(* CODESYS project CAN API.library
   Author: 3S - Smart Software Solutions GmbH
   Title: CAN API
   Version: 1.0.0.3
   DocFormat: reStructuredText
   Description: This library provides an easy to use interface for sending and receiving CAN messages. The library is optimized for Structured Text and graphical (CFC) programming.
   Company: 3S - Smart Software Solutions GmbH
   LanguageModelAttribute: qualified-access-only
   DefaultNamespace: CAN

Project tree, tasks and I/O mapping:
  libraries: CAA Behaviour Model, * (CAA Technical Workgroup); CANbus, * (3S - Smart Software Solutions GmbH); CAA Memory Block Manager Extern, * (CAA Technical Workgroup); Standard, * (System)
  Enums/
    data type RECEIVERTYPE
    data type BUSSTATE
    data type ERROR
  Interfaces/
    interface IMessageProcessor: ProcessMessage
    interface ICANBus29bit
    interface ICANDriver: ICANBus
    interface ICANBusBase: GetBusDiagnosis, DeleteReceiver, GetAreaReceiver, ReceiveMessage, SendMessage, ResetBusAlarm, CloseCANDriver, Is29bit, GetMaskReceiver, GetSingleIdReceiver
    interface ICANBus11bit
  00000000-0000-0000-0000-000000000000|D:\CoDeSys\LibrariesV3\trunk\Intern\CAA\CAA Template\3.4.0.0 draft\Placeholder.xml
  00000000-0000-0000-0000-000000000000|D:\CoDeSys\LibrariesV3\trunk\Intern\CAA\CAA Template\3.2.0.3 draft\Prefix.pdf
  Function Blocks/
    Object Oriented Programming/
      function block CANBus_11bit [ST]: GetBusDiagnosis, Is29bit, ResetBusAlarm, ReceiveMessage, CloseCANDriver, DeleteReceiver, GetMaskReceiver, GetAreaReceiver, GetSingleIdReceiver, SendMessage
      function block CANBus_Base [ST]: CloseCANDriver, SendMessage, DeleteReceiver, FreeReceiverBlock, ReceiveAlwaysNewest, GetReceiverBlock, CreateMaskReceiver, CreateAreaReceiver, ReceiveQueued, CreateSingleIDReceiver, CreateDriver, BusAlarm, GetAreaReceiver, GetMaskReceiver, ReceiveMessage, FB_Init, GetBusDiagnosis, ResetBusAlarm, Is29bit, GetSingleIdReceiver
      function block CANBus_29bit [ST]: ResetBusAlarm, SendMessage, DeleteReceiver, GetMaskReceiver, ReceiveMessage, Is29bit, CloseCANDriver, GetAreaReceiver, GetBusDiagnosis, GetSingleIdReceiver
    Graphical Programming/
      function block CANSender [ST]: prvAbort, prvResetOutputs, prvStart, prvCyclicAction
      function block CANBusDiagnosis [ST]: prvResetOutputs, prvCyclicAction, prvStart, prvAbort
      function block CANDriver_11bit [ST]: ICANBus, prvCyclicAction, prvAbort, prvStart, prvResetOutputs
      function block CANAreaReceiver [ST]: prvAbort, prvCyclicAction, prvResetOutputs, prvStart
      function block CANDriver_29bit [ST]: ICANBus, prvCyclicAction, prvResetOutputs, prvStart, prvAbort
      function block CANMaskReceiver [ST]: prvStart, prvAbort, prvCyclicAction, prvResetOutputs
      function block CANSingleIdReceiver [ST]: prvResetOutputs, prvStart, prvAbort, prvCyclicAction
  Structs/
    data type RECEIVER_INFO
    data type DRIVER_CONFIG
    data type RECEIVER_MASK
    data type MESSAGE
    data type RxMESSAGE
    data type RECEIVER_AREA
    data type DIAGNOSIS_INFO
    data type RECEIVER_SINGLE_ID
*)

// Structs/RECEIVER_INFO
{attribute 'hide'}
{attribute 'qualified_only'}
TYPE RECEIVER_INFO :
STRUCT
	hReceiver : CAA.HANDLE;
	eType : RECEIVERTYPE;
END_STRUCT
END_TYPE

// Structs/DRIVER_CONFIG
/// This data type describes the configuration of a CANbus Driver
{attribute 'qualified_only'}
TYPE DRIVER_CONFIG :
STRUCT
	uiBaudrate 		: UINT; (* Possible values for baud rate [kbit/s]: 10, 20, 50, 100, 125, 250, 500, 800 or 1000. *)
	usiNetwork 		: USINT; (* number of the interface (Network ID starts by 0) *)
	ctMessages		: USINT; (* length of the message queue for outgoing messages *)
END_STRUCT
END_TYPE

// Structs/RECEIVER_MASK
/// | The parameter canIdMask describes a bit mask for canId’s on incoming messages. 
/// | The parameter canIdValue proofs if the mask applies to the CanId of the received message. 
/// | If the CanId doesn’t apply to the mask, the message will be filtered out. 
/// | For the use of the other Mask/Value parameters see the examples of RECEIVER_AREA.
{attribute 'qualified_only'}

TYPE RECEIVER_MASK :
STRUCT
	dwIdValue 			: DWORD; (* bit sign of identifier of message *)
	dwIdMask 			: DWORD; (* mask for bit sign of IdValue *)
	xRTRValue 			: BOOL; (* bit sign for RTR flag *)
	xRTRMask 			: BOOL; (* mask for bit sign of xRTRValue  *)
	x29BitIdValue 		: BOOL; (* 29-Bit message *)
	x29BitIdMask 		: BOOL; (* Mask for 29-bit message *)
	xTransmitValue 		: BOOL; (* Messages sent via this adapter with the same driver. *)
	xTransmitMask 		: BOOL; (* Mask for messages sent via this adapter with the same driver. *)
	xAlwaysNewest 		: BOOL; (* TRUE: only the most current message will be received; FALSE: all messages will be received *)
END_STRUCT
END_TYPE

// Enums/RECEIVERTYPE
/// | This data type distinguishes if a receiver receives always the newest message or not  
{attribute 'qualified_only'}
TYPE RECEIVERTYPE :
(
	QUEUED_RECEIVER, (* receiving all messages *)
	ALWAYS_NEWEST_RECEIVER (* receiving only the newest message *)
) BYTE;
END_TYPE

// Enums/BUSSTATE
/// | This data type describes the current state of the CAN network.
{attribute 'qualified_only'}
TYPE BUSSTATE :
(
	UNKNOWN := 0, (* The state of the network is not known. Its functionality is not implemented. *)
	ERR_FREE, (* No occurrence of CAN bus errors so far. The error counters of the chip are zero. *)
	ACTIVE, (* Only few CAN bus errors so far. The error counters of the chip are below the warning level. *)
	WARNING, (* Occurrence of some CAN bus errors. The error counters are above the warning level. *)
	PASSIVE, (* Too many CAN bus errors. The error counters are above the error level. *)
	BUSOFF (* The node has been separated from the CAN bus. The error counter has exceeded the admissible maximum. *)
)BYTE;
END_TYPE

// Structs/MESSAGE
/// | This structure contains the information of a message. 
/// | Messages of this type can be sent via CANSender (FB) in CFC or by an instance of CANBus_11bit / CANBus_29bit  
/// | in ST programs.
{attribute 'qualified_only'}
TYPE MESSAGE :
STRUCT
	udiCanID 		: UDINT; (* CAN-ID (Communication Object Identifier) is the bitId of a CAN-frame *)
	abyData 		: ARRAY[0..7] OF BYTE; (* Array for 0 to 7 bytes of data *)
	usiDataLength 	: USINT; (* The length of the data array 0 to 8 *)
	xRTR 			: BOOL; (* Remote Transmission Request *)
	xIs29BitMessage	: BOOL; (* TRUE: the messages is a 29bit message, FALSE: the message is a 11bit message *)
END_STRUCT
END_TYPE

// Structs/RxMESSAGE
/// | The structure of a received message. RxMESSAGE has two more elements as MESSAGE.
/// | Messages of the type RxMESSAGE can be used the same way as messages of the type MESSAGE
{attribute 'qualified_only'}
TYPE RxMESSAGE EXTENDS MESSAGE :
STRUCT
		xIsTxMessage	: BOOL := TRUE; (* TRUE: Messages sent via this adapter with the same driver. *)
		udiTSP			: UDINT; (* Only available if the driver supports TimeStamps. If not the value is 0. Compare TimeStamp by calling SysTimeGetUs() function *)
END_STRUCT
END_TYPE

// Structs/RECEIVER_AREA
/// | This structure identifies an area for receiving CANBus frames. 
/// | Please note that the Area Receiver only allows 11bit CAN-IDs. If the mask parameter is TRUE, 
/// | a filter in the CAN Receiver Queue is active. 
/// | Now messages are filtered according to the value parameter. 
/// |
/// | Examples:
/// | Only Transmit messages ranging between 16#100 and 16#150: 
/// | dwIdStart:=16#100, dwIdEnd:=16#150, xTransmitValue = TRUE, xTransmitMask = TRUE, all other Mask paramters = FALSE
/// |
/// | All messages ranging between 16#0 and 16#7FF 
/// | dwIdStart:=16#0, dwIdEnd:=16#7FF all mask parameters FALSE (no further filtering is done).
/// |
/// | All messages: dwIdStart = 0, dwIdEnd = 0, 
/// | all Mask Parameter FALSE all Value Parameter FALSE
/// |
{attribute 'qualified_only'}
TYPE RECEIVER_AREA :
STRUCT
	dwIdStart		: DWORD; (* first identifier of the area *)
	dwIdEnd			: DWORD; (* last identifier of the area *)
	xRTRValue		: BOOL; (* bit sign for RTR flag *)
	xRTRMask		: BOOL; (* mask for bit sign of xRTRValue  *)
	xTransmitValue	: BOOL; (* Messages sent via this adapter with the same driver. *)
	xTransmitMask	: BOOL; (* Mask for messages sent via this adapter with the same driver. *)
END_STRUCT
END_TYPE

// Structs/DIAGNOSIS_INFO
/// This data type describes diagnostic information 
{attribute 'qualified_only'}
TYPE DIAGNOSIS_INFO :
STRUCT
	ctSendCounter			: CAA.COUNT; (* The value of the send counter. *)
	ctReceiveCounter		: CAA.COUNT; (* The value of the receive counter. *)
	ctRxErrorCounter		: CAA.COUNT; (* The value of the receive error counter. *)
	ctTxErrorCounter		: CAA.COUNT; (* The value of the send error counter. *)	
	ctLostCounter			: CAA.COUNT; (* The value of the lost messages. *)
	ctReceivePoolSize		: CAA.COUNT; (* Size of the receive pool *)
	ctReceiveQueueLength	: CAA.COUNT; (* Size of the receive queue length *)
	ctTransmitPoolSize		: CAA.COUNT; (* Size of the transmit pool *)
	ctTransmitQueueLength	: CAA.COUNT; (* Size of the transmit queue length *)
	xBusAlarm				: BOOL; (* Bus Alarm *)
	usiBusLoad				: USINT; (* The bus load. *)
	xSendingActive			: BOOL; (*  TRUE: the CAN hardware is busy sending CAN messages. FALSE: all messages have already been sent. *)
	eState					: BUSSTATE; (* This data type describes the state of the CAN network. *)
	uiBaudrate				: UINT; (* The baud rate of the bus. *)
END_STRUCT
END_TYPE

// Enums/ERROR
/// | This data type describes errors
{attribute 'qualified_only'}
TYPE ERROR : 
(
		NO_ERROR := 0, (* No error occurred *)
		INTERNAL_ERROR, (* An error occurred in the CL2 Library. Please check with brake points. *)
		NO_MEMORY, (* no more memory *)
		NO_CANBUS_DRIVER, (* Create a valid CANBus Driver for this operation *)
		NO_VALID_RECEIVER, (* There is no valid receiver *)
		START_VALUE_GT_END, (* Start value is greater than end value for area receiver *)
		TIME_OUT, (* Time out *)
		BUS_ALARM, (* The CAN Bus is in alarm state *)
		MESSAGE_QUEUE_EXCEEDED, (* The sending queue is full *)
		ONLY_11BIT_CANID_ALLOWED, (* CAN-IDs needs to be max. 11bit *)
		WRONG_BAUDRATE, (* Baudrate for CANDriver is not valid *)
		WRONG_PARAMETER, (* A parameter has a wrong value *)
		CANBUS_DRIVER_NOT_CREATED (* NetID might be wrong or the driver is not registered in "GatewayPLC/CoDeSysControl.cfg".
									Example 1: 1 CAN card with 2 channels, channel 1: NetId = 0, channel 2: NetId = 1;
									Example 2: 2 CAN cards: NetId depends on the order the drivers are loaded. *) 
)BYTE; 
END_TYPE

// Structs/RECEIVER_SINGLE_ID
/// | This structure filters the messages of a single CAN Id. 
/// | If the mask parameter is TRUE, a filter in the CAN Receiver Queue is active. 
/// | Now messages are filtered according to the value parameter. Also see the examples of RECEIVER_AREA.
{attribute 'qualified_only'}
TYPE RECEIVER_SINGLE_ID :
STRUCT
	dwCanId			: DWORD; (* CanId *)
	xRTRValue		: BOOL; (* bit sign for RTR flag *)
	xRTRMask		: BOOL; (* mask for bit sign of xRTRValue  *)
	x29BitIdValue	: BOOL; (* 29-Bit message *)
	x29BitIdMask	: BOOL; (* Mask for 29-bit message *)
	xTransmitValue	: BOOL; (* Messages sent via this adapter with the same driver. *)
	xTransmitMask	: BOOL; (* Mask for messages sent via this adapter with the same driver. *)
	xAlwaysNewest	: BOOL; (* TRUE: only the most current message will be received; FALSE: all messages will be received *)
END_STRUCT
END_TYPE

// Interfaces/IMessageProcessor
/// All received messages are passed to the MessageProcessor. The method ProcessMessage() must be implemented by the user.
INTERFACE IMessageProcessor

/// | The Process Message Method must be implemented by the user.
/// | Define here how you wish to proceed with incoming messages.
METHOD ProcessMessage
VAR_IN_OUT
	Message 		: RxMESSAGE; (* Incoming message *)
END_VAR
END_METHOD

END_INTERFACE

// Interfaces/ICANBus29bit
{attribute 'hide'}
INTERFACE ICANBus29bit EXTENDS ICANBusBase

END_INTERFACE

// Interfaces/ICANBusBase
{attribute 'hide'}
INTERFACE ICANBusBase EXTENDS __SYSTEM.IQueryInterface

METHOD GetBusDiagnosis : BOOL
VAR_IN_OUT
	DiagnosticInfo		: DIAGNOSIS_INFO; (* This data type descripes diagnostic information  *)
END_VAR
VAR_OUTPUT
	eError				: ERROR; (* Error codes *)
END_VAR
END_METHOD

METHOD DeleteReceiver : BOOL
VAR_IN_OUT
	hReceiver		: CAA.HANDLE; (* Receiver to be deleted *)
END_VAR
VAR_OUTPUT
	eError			: ERROR; (* Error codes *)
END_VAR
END_METHOD

METHOD GetAreaReceiver : CAA.HANDLE
VAR_IN_OUT
	Area				: RECEIVER_AREA; (* Structure with the information of the bit masks and a range of CAN-IDs *)
END_VAR
VAR_OUTPUT
	eError				: ERROR; (* Error codes *)
END_VAR
END_METHOD

METHOD ReceiveMessage : BOOL
VAR_INPUT
	hReceiver 		: CAA.HANDLE; (* Eather a MaskReceiver or AreaReceiver *)
	itfMsgProcessor : IMessageProcessor;
	tTimeLimit		: TIME;
END_VAR
VAR_OUTPUT
	eError			: ERROR; (* Error codes *)
END_VAR
END_METHOD

METHOD SendMessage : BOOL
VAR_IN_OUT
	Message 		: Message; (* Structure with the frame information and data to be sent. *)
END_VAR
VAR_OUTPUT
	eError			: ERROR; (* Error codes *)
END_VAR
END_METHOD

METHOD ResetBusAlarm : BOOL
VAR_INPUT
END_VAR
VAR_OUTPUT
	eError			: ERROR; (* Error codes *)
END_VAR
END_METHOD

METHOD CloseCANDriver : BOOL
VAR_OUTPUT
	eError			: ERROR; (* Error codes *)
END_VAR
END_METHOD


PROPERTY Is29bit : BOOL
GET
END_GET
END_PROPERTY

METHOD GetMaskReceiver : CAA.HANDLE
VAR_IN_OUT
	Mask				: RECEIVER_MASK; (* Structure with the information of the bit masks *)
END_VAR
VAR_OUTPUT
	eError				: ERROR; (* Error codes *)
END_VAR
END_METHOD

METHOD GetSingleIdReceiver : CAA.HANDLE
VAR_IN_OUT
	SingleId			: RECEIVER_SINGLE_ID; (* Structure with the information of the bit masks *)
END_VAR
VAR_OUTPUT
	eError				: ERROR; (* Error codes *)
END_VAR
END_METHOD

END_INTERFACE

// Function Blocks/Graphical Programming/CANSender
/// | CANSender will send messages over a CANDriver. It is possible to send frames with 29 bit and 11 bit frames. 
/// | This depends on the CAN Driver used for instantiating the CAN Sender. A CAN Sender instantiated with a 29BitCANDriver 
/// | is able to send 11 bit messages as well as 29 bit messages. The sending method is defined by 
/// | setting the xSendAs29bitMsg flag of MESSAGE. An 11BitCANDriver can only send 11 bit messages. 
/// | If CANSender uses an 11bit driver xSendAs29bitMsg of MESSAGE will be ignored.
FUNCTION_BLOCK CANSender EXTENDS CBM.ETrig
VAR_INPUT
	itfCANDriver	: ICANDriver; (* Messages are sent with this driver *)
END_VAR
VAR_IN_OUT
	Message 		: MESSAGE; (* Message information and data. *)
END_VAR
VAR_OUTPUT
	eError			: ERROR; (* Error codes *)
END_VAR
VAR
	_itf11bit			: ICANBus11bit;
	_itf29bit			: ICANBus29bit;
	_hReceiver			: CAA.HANDLE;
	_pMessage 			: POINTER TO MESSAGE;
END_VAR

_pMessage := ADR(Message);
SUPER^();

{attribute 'hide'}
METHOD prvAbort : BOOL
VAR_INPUT
END_VAR
VAR
END_VAR
(*IF xError THEN (* abort because of error *)

ELSE (* user abort *)

END_IF*)
xAbortInProgress:= FALSE;
END_METHOD

{attribute 'hide'}
METHOD prvResetOutputs : BOOL
VAR_INPUT
END_VAR
VAR
END_VAR
eError:= ERROR.NO_ERROR;
SUPER^.prvResetOutputs();
END_METHOD

{attribute 'hide'}
METHOD prvStart : BOOL
VAR_INPUT
END_VAR
VAR
END_VAR
END_METHOD

{attribute 'hide'}
METHOD prvCyclicAction : BOOL
VAR_INPUT
END_VAR
VAR
END_VAR
IF _pMessage <> CAA.gc_pNULL THEN
	IF (itfCANDriver.ICANBus.Is29bit) THEN
		__QUERYINTERFACE(itfCANDriver.ICANBus, _itf29Bit);
		_itf29bit.SendMessage(Message:=_pMessage^, eError=>eError);
	ELSE
		__QUERYINTERFACE(itfCANDriver.ICANBus, _itf11Bit);
		_itf11bit.SendMessage(Message:=_pMessage^, eError=>eError);
	END_IF
END_IF

IF eError = ERROR.NO_ERROR THEN
	xDone:= TRUE;
ELSE
	iError:= 2;
END_IF
END_METHOD

END_FUNCTION_BLOCK

// Interfaces/ICANDriver
/// | CANDriver_11bit and CANDriver_29bit implement this interface. 
/// | CANSender, CANMaskReceiver, CANAreaReceiver and CANBusDiagnosis expect a CANDriver instance that implements 
/// | the ICANDriver interface.
INTERFACE ICANDriver

{attribute 'hide'}
PROPERTY ICANBus : ICANBusBase
GET
END_GET
END_PROPERTY

END_INTERFACE

// Function Blocks/Graphical Programming/CANDriver_11bit
/// | This CAN Driver can handle frames with 11bit CAN-IDs. If a CAN Sender gets instantiated with this Driver all messages
/// | are sent in 11 bit frames. The xSendAs29bitMsg flag of Message will be ignored. Any Receiver instantiated with this Driver
/// | will only receive frames with 11 bit CAN-IDs. In case of a Bus Alarm it’s possible to reset the driver through xResetBusAlarm.
FUNCTION_BLOCK CANDriver_11bit EXTENDS CBM.LTrig IMPLEMENTS ICANDriver
VAR_INPUT
	xResetBusAlarm	: BOOL; (* TRUE: Reset the Bus Alarm (applies only if the Bus Driver is in alarm state). *)
END_VAR
VAR_IN_OUT
	DriverConfig	: DRIVER_CONFIG; (* Information to setup the CANbus Driver *)
END_VAR
VAR_OUTPUT
	xBusAlarm		: BOOL; (* Indicates if a Bus Alarm occurred *)
	eError			: ERROR; (* Error codes *)
END_VAR
VAR
	_CANBus			: CANBus_11bit;
	_pDriverConfig	: POINTER TO DRIVER_CONFIG;
END_VAR

_pDriverConfig := ADR(DriverConfig);
SUPER^();
IF iError = CBM.ERROR.TIME_OUT THEN
	eError := ERROR.TIME_OUT;
END_IF

{attribute 'hide'}
PROPERTY ICANBus : ICANBusBase
GET
ICANBus:= _CANBus;
END_GET
END_PROPERTY

{attribute 'hide'}
METHOD prvCyclicAction : BOOL
VAR_INPUT
END_VAR
VAR
END_VAR
IF xEnable AND _pDriverConfig <> CAA.gc_pNULL THEN
	_CANBus(DriverConfig:= _pDriverConfig^, eError=> eError);
	IF _CANBus.BusAlarm THEN 
		eError:= ERROR.BUS_ALARM;
		xBusAlarm:= TRUE;
	ELSIF (*_CANBus.BusAlarm AND*) xResetBusAlarm  THEN
		_CANBus.ResetBusAlarm(eError=> eError);
		xBusAlarm:= FALSE;
	END_IF
END_IF

IF eError <> ERROR.NO_ERROR THEN
	iError:= 2;
END_IF
END_METHOD

{attribute 'hide'}
METHOD prvAbort : BOOL
VAR_INPUT
END_VAR
VAR
END_VAR
IF xError THEN (* abort because of error *)
	_CANBus.CloseCANDriver(eError=> eError);
ELSE
	_CANBus.CloseCANDriver(eError=> eError);
END_IF
xAbortInProgress:= FALSE;
END_METHOD

{attribute 'hide'}
METHOD prvStart : BOOL
VAR_INPUT
END_VAR
VAR
END_VAR
END_METHOD

{attribute 'hide'}
METHOD prvResetOutputs : BOOL
VAR_INPUT
END_VAR
VAR
END_VAR
eError:= ERROR.NO_ERROR;
xBusAlarm:= FALSE;
SUPER^.prvResetOutputs();
END_METHOD

END_FUNCTION_BLOCK

// Function Blocks/Object Oriented Programming/CANBus_11bit
/// | CANBus_11bit can handle frames with 11bit CAN-IDs. An instance of this function block has to be created in order 
/// | for being able to send or receive messages. The FB expects a complete structure of the type DRIVER_CONFIG 
/// | to set up the CANBus.
FUNCTION_BLOCK CANBus_11bit EXTENDS CANBus_Base IMPLEMENTS ICANBus11bit
VAR_INPUT
END_VAR
VAR_OUTPUT
END_VAR
VAR
END_VAR

/// Call of the CANBus_Base FB
SUPER^._x29bitSupport:= FALSE;
SUPER^();

/// This method aggregates diagnostic information in DIAGNOSIS_INFO 
METHOD GetBusDiagnosis : BOOL
VAR_IN_OUT
	DiagnosticInfo		: DIAGNOSIS_INFO; (* This data type descripes diagnostic information  *)
END_VAR
VAR_OUTPUT
	eError				: ERROR; (* Error codes *)
END_VAR
/// Method call of the CANBus_Base FB
GetBusDiagnosis:= SUPER^.GetBusDiagnosis(DiagnosticInfo:= DiagnosticInfo, eError=> eError);
END_METHOD

{attribute 'hide'}
PROPERTY Is29bit : BOOL
GET
Is29bit:= FALSE;
END_GET
END_PROPERTY

/// This method resets the CANBus if the driver is in 'bus alarm' state. 
METHOD ResetBusAlarm : BOOL
VAR_INPUT
END_VAR
VAR_OUTPUT
	eError			: ERROR; (* Error codes *)
END_VAR
/// Method call of the CANBus_Base FB
ResetBusAlarm:= SUPER^.ResetBusAlarm(eError=> eError);
END_METHOD

/// | ReceiveMessage expects a valid handle to either an AreaReceiver, SingleIdReceiver or a MaskReceiver. 
/// | With receivers it is possible to filter incoming messages. If a time limit is set, the receiver will 
/// | receive in each cycle messages until the time is up. It there is no time limit set (tTimeLimit:= 0), 
/// | the receiver receives messages until the receiver buffer is empty. If the time limit is too small it 
/// | may be that not all received messages are processed and therefor the buffer gets smaller until there 
/// | are no free message handles left. Received messages will be passed to the Message Processor. All message 
/// | information will be available there. The Message Processor must be implemented by the user.
METHOD ReceiveMessage : BOOL
VAR_INPUT
	hReceiver 		: CAA.HANDLE; (* Either a MaskReceiver, SingleIdReceiver or AreaReceiver *)
	itfMsgProcessor : IMessageProcessor; (* The Message Processor will process the read messages accrding to the implementation of the user *)
	tTimeLimit		: TIME; (* The time limit for reading messages. (T#0s means no time limit) *)
END_VAR
VAR_OUTPUT
	eError			: ERROR; (* Error codes *)
END_VAR
/// Method call of the CANBus_Base FB
ReceiveMessage:= SUPER^.ReceiveMessage(hReceiver:= hReceiver, itfMsgProcessor:= itfMsgProcessor, tTimeLimit:= tTimeLimit, eError=> eError);
END_METHOD

/// | Closes the CAN Driver. After closing, messages can't be received or transmitted anymore.
METHOD CloseCANDriver : BOOL
VAR_INPUT
END_VAR
VAR_OUTPUT
	eError			: ERROR; (* Error codes *)
END_VAR
CloseCANDriver:= SUPER^.CloseCANDriver(eError=> eError);
END_METHOD

/// Deletes given receiver
METHOD DeleteReceiver : BOOL
VAR_IN_OUT
	hReceiver		: CAA.HANDLE; (* Receiver to be deleted *)
END_VAR
VAR_IN_OUT
END_VAR
VAR_OUTPUT
	eError			: ERROR; (* Error codes *)
END_VAR
/// Method call of the CANBus_Base FB
DeleteReceiver:= super^.DeleteReceiver(hReceiver:= hReceiver, eError=> eError);
END_METHOD

/// | Creates a mask for receiving messages. (With each call of this function a Receiver is created. 
/// | Therefor the method should not be called cyclic.)
METHOD GetMaskReceiver : CAA.HANDLE
VAR_IN_OUT
	Mask				: RECEIVER_MASK; (* Structure with the information of the bit masks *)
END_VAR
VAR_OUTPUT
	eError				: ERROR; (* Error codes *)
END_VAR
/// Method call of the CANBus_Base FB
GetMaskReceiver:= SUPER^.GetMaskReceiver(Mask:= Mask, eError=> eError);
END_METHOD

/// | Creates a receiver to receive messages within a range of CAN-IDs. 
/// | (With each call of this function a Receiver is created. Therefor the method should not be called cyclic.)
METHOD GetAreaReceiver : CAA.HANDLE
VAR_IN_OUT
	Area				: RECEIVER_AREA; (* Structure with the information of the bit masks and a range of CAN-IDs *)
END_VAR
VAR_OUTPUT
	eError				: ERROR; (* Error codes *)
END_VAR
/// Method call of the CANBus_Base FB
GetAreaReceiver:= SUPER^.GetAreaReceiver(Area:= Area, eError=> eError);
END_METHOD

/// | Generates a receiver for filtering a single CanId. (With each call of this function a 
/// | Receiver is created. Therefor the method should not be called cyclic.)
METHOD GetSingleIdReceiver : CAA.HANDLE
VAR_IN_OUT
	(* Structure with the information of the bit masks *)
	SingleId	: RECEIVER_SINGLE_ID;
END_VAR
VAR_OUTPUT
	(* Error codes *)
	eError	: ERROR;
END_VAR
/// Method call of the CANBus_Base FB
GetSingleIdReceiver:= SUPER^.GetSingleIdReceiver(SingleId:= SingleId, eError=> eError);
END_METHOD

/// Send a message. If the message got sent the return value is true.
METHOD SendMessage : BOOL
VAR_IN_OUT
	Message 		: MESSAGE; (* Message information and data. *)
END_VAR
VAR_OUTPUT
	eError			: ERROR; (* Error codes *)
END_VAR
SendMessage := SUPER^.SendMessage(Message := Message, eError => eError);
END_METHOD

END_FUNCTION_BLOCK

// Function Blocks/Object Oriented Programming/CANBus_Base
/// This is the base function block for CANBus_11bit and CANBus_29bit
{attribute 'hide'}
FUNCTION_BLOCK CANBus_Base IMPLEMENTS ICANBusBase
VAR_INPUT
	DriverConfig	: DRIVER_CONFIG; (* This structure contains the informaiton for creating a CANbus Driver *)
END_VAR
VAR_OUTPUT
	eError			: ERROR; (* Error codes *)
END_VAR
VAR
	_hDriver			: CAA.HANDLE; (* The handle for the CANbus Driver *)
	_hReceiverPool		: CAA.HANDLE;
	_x29bitSupport	: BOOL;
	_eErrorInternal	: CL2.ERROR; (* error codes from the CL2 library *)
END_VAR

/// By calling the private method CreateDriver() a CANbus Driver will be created. The driver is accessable through hDriver.
IF _hDriver = CAA.gc_hINVALID THEN
	CreateDriver(DriverConfig:= DriverConfig, x29bitSupport:= _x29bitSupport, hDriver=> _hDriver, eError=> eError);
END_IF

/// Closes the CAN Driver. After closing, messages can't be received or transmitted anymore.
METHOD CloseCANDriver : BOOL
VAR_INPUT
END_VAR
VAR_OUTPUT
	eError			: ERROR; (* Error codes *)
END_VAR
VAR
	eErrorInternal	: CL2.ERROR; (* error codes from the CL2 library *)
END_VAR
IF _hDriver <> CAA.gc_hINVALID THEN
	eErrorInternal:= CL2.DriverClose(hDriver:= _hDriver);
	IF eErrorInternal <> CL2.ERROR.NO_ERROR THEN
		eError:= ERROR.INTERNAL_ERROR;
	ELSE
		_hDriver:= CAA.gc_hINVALID;
		CloseCANDriver:= TRUE;
	END_IF
ELSE
	eError:= ERROR.NO_CANBUS_DRIVER;
END_IF
END_METHOD

/// Send a message. If the message got sent the return value is true.
METHOD SendMessage : BOOL
VAR_IN_OUT
	Message 		: MESSAGE; (* Message information and data. *)
END_VAR
VAR_OUTPUT
	eError			: ERROR; (* Error codes *)
END_VAR
VAR
	hMessage		: CAA.HANDLE; (* Pointer to the created Message *)
	eErrorInternal	: CL2.ERROR; (* error codes from the CL2 library *)
	pData			: POINTER TO CL2i.DATA; (* Pointer to the data array of the created message *)
	i				: INT; (* Counter *)
END_VAR
IF(_hDriver <> CAA.gc_hINVALID)THEN
	IF NOT Is29Bit AND MESSAGE.xIs29BitMessage THEN
		eError := ERROR.ONLY_11BIT_CANID_ALLOWED;
		RETURN;
	END_IF
	
	IF NOT Message.xIs29BitMessage THEN
		IF Message.udiCanID > 16#7FF THEN
			eError := ERROR.WRONG_PARAMETER;
			RETURN;
		END_IF
	END_IF
	
	/// First it creates a new message with the data from Message by calling CL2.CreateMessage()
	hMessage:= CL2.CreateMessage(
				hDriver:= _hDriver, 
				cobID:= Message.udiCanId, 
				usiLength:= Message.usiDataLength, 
				xRTR:= Message.xRTR, 
				x29BitID:= Message.xIs29BitMessage,
				peError:= ADR(eErrorInternal));

	IF hMessage <> CAA.gc_hINVALID THEN
		IF Message.usiDataLength > 0 THEN
			/// The data from the data-array will be copied into the data-array of the created message			
			pData:= CL2.GetMessageDataPointer(hMessage:= hMessage, peError:= ADR(eErrorInternal));
			FOR i:=0 TO Message.usiDataLength -1 DO
				pData^[i]:= Message.abyData[i];
			END_FOR
		END_IF
		
		/// The frame with the data is sent when CL2.Write() gets called.			
		eErrorInternal := CL2.Write(hDriver:= _hDriver, hMessage:= hMessage, usiPriority:= 2, xEnableSyncWindow:= FALSE);
		IF eErrorInternal <> CL2.ERROR.NO_ERROR THEN
			eError:= ERROR.INTERNAL_ERROR;
			IF hMessage <> CAA.gc_hINVALID THEN
				CL2.FreeMessage(hMessage:= hMessage);
				hMessage := CAA.gc_hINVALID;
			END_IF
		ELSE
			SendMessage:= TRUE;
		END_IF
	ELSE
		eError:= ERROR.MESSAGE_QUEUE_EXCEEDED;
	END_IF
ELSE
	eError:= ERROR.NO_CANBUS_DRIVER;
END_IF
END_METHOD

/// Deletes any receiver
METHOD DeleteReceiver : BOOL
VAR_IN_OUT
	hReceiver		: CAA.HANDLE; (* Receiver to be deleted *)
END_VAR
VAR_IN_OUT
END_VAR
VAR_OUTPUT
	eError			: ERROR; (* Error codes *)
END_VAR
VAR
	pReceiverInfo : POINTER TO RECEIVER_INFO;
	eErrorInternal	: CL2.ERROR; (* error codes from the CL2 library *)
	eMBMError : MBM.ERROR;
END_VAR
IF hReceiver <> CAA.gc_hINVALID THEN
	pReceiverInfo := MBM.BlockGetData(hBlock := hReceiver, peError := ADR(eMBMError));
	IF pReceiverInfo <> CAA.gc_pNULL THEN
		eErrorInternal:= CL2.DeleteReceiver(hReceiverId:= pReceiverInfo^.hReceiver);
		pReceiverInfo^.hReceiver := CAA.gc_hINVALID;
		MBM.PoolPutBlock(hReceiver);
		DeleteReceiver:= TRUE;
	ELSE
		eError:= ERROR.NO_VALID_RECEIVER;
	END_IF
ELSE
	eError:= ERROR.NO_VALID_RECEIVER;
END_IF
END_METHOD

METHOD PRIVATE FreeReceiverBlock
VAR_INPUT
	hReceiverBlock : CAA.HANDLE;
END_VAR
VAR
END_VAR
MBM.PoolPutBlock(hBlock := hReceiverBlock);
END_METHOD

METHOD PRIVATE ReceiveAlwaysNewest : BOOL
VAR_INPUT	
	hReceiver 		: CAA.HANDLE; (* Eather a MaskReceiver or AreaReceiver *)
	itfMsgProcessor : IMessageProcessor; (* The Message Processor will process the read messages accrding to the implementation of the user *)
END_VAR
VAR_OUTPUT
	eError			: ERROR; (* Error codes *)
END_VAR
VAR
	eErrorInternal	: CL2.ERROR; (* error codes from the CL2 library *)
	hMessage		: CAA.HANDLE := CAA.gc_hINVALID; (* Handle for an incoming message *)
	Message			: RxMESSAGE;
	pData			: POINTER TO CL2i.DATA; (* Pointer to the data-array of the incoming message *)
	ctMsgLeft		: CAA.COUNT; (* Counter of the messages left in the queue *)
	i				: INT; (* counter variable *)
	udiTSP			: UDINT; (* Only if the driver supports TimeStamps. If not the value is 0. Compare TimeStamp by calling SysTimeGetUs() function *)
END_VAR
hMessage:= CL2.Read(hReceiverID:= hReceiver, pctMsgLeft:= ADR(ctMsgLeft), peError:= ADR(eErrorInternal));
IF hMessage <> CAA.gc_hINVALID THEN
	IF ctMsgLeft > 0 THEN
		/// If a message was received the frame information and the data-array will be written into Message.
		Message.udiCanId:= CL2.GetMessageId(hMessage:= hMessage, peError:= ADR(eErrorInternal));
		Message.usiDataLength:= CL2.GetMessageLength(hMessage:= hMessage, peError:= ADR(eErrorInternal));
		Message.xRTR:= CL2.IsRTRMessage(hMessage:= hMessage, peError:= ADR(eErrorInternal));
		Message.xIs29BitMessage:= CL2.Is29BitIdMessage(hMessage:= hMessage, peError:= ADR(eErrorInternal));
		Message.xIsTxMessage:= CL2.IsTransmitMessage(hMessage:= hMessage, peError:= ADR(eErrorInternal));
		udiTSP:= CL2.GetTimeStamp(hMessage:= hMessage, peError:= ADR(eErrorInternal));
		IF Message.usiDataLength > 0 THEN
			pData:= CL2.GetMessageDataPointer(hMessage:= hMessage, peError:= ADR(eErrorInternal));	
		
			IF (pData <> CAA.gc_pNULL) THEN
				FOR i:= 0 TO Message.usiDataLength - 1 DO
					Message.abyData[i] := pData^[i];
				END_FOR
			END_IF
		END_IF
		
		/// The received message will be processed by the Message Processor
		itfMsgProcessor.ProcessMessage(Message:= Message);
		ReceiveAlwaysNewest := TRUE;
	END_IF
	
	/// When finished processing the data the memory for the message handle hMessage will be freed by calling CL2.FreeMessage()		
	CL2.FreeMessage(hMessage := hMessage);
ELSIF eErrorInternal <> CL2.ERROR.NO_ERROR THEN
	eError:= ERROR.INTERNAL_ERROR;
END_IF
END_METHOD

METHOD PRIVATE GetReceiverBlock : CAA.HANDLE
VAR_INPUT
	peError : POINTER TO ERROR;
END_VAR
VAR_OUTPUT
	pReceiverInfo : POINTER TO RECEIVER_INFO;
END_VAR
VAR
	hReceiverInfo		: CAA.HANDLE;
	eMBMError 			: MBM.ERROR;
END_VAR
hReceiverInfo := MBM.PoolGetBlock(hPool := _hReceiverPool, peError := ADR(eMBMError));
IF hReceiverInfo = CAA.gc_hINVALID THEN
	MBM.PoolExtendH(hPool := _hReceiverPool, 10);
	hReceiverInfo := MBM.PoolGetBlock(hPool := _hReceiverPool, peError := ADR(eMBMError));
END_IF

IF eMBMError <> MBM.ERROR.NO_ERROR OR hReceiverInfo = CAA.gc_hINVALID THEN
	IF peError <> CAA.gc_pNULL THEN
		peError^ := ERROR.NO_MEMORY;
	END_IF
ELSE
	pReceiverInfo := MBM.BlockGetData(hBlock := hReceiverInfo, peError := ADR(eMBMError));
END_IF

GetReceiverBlock := hReceiverInfo;
END_METHOD

/// Create a Mask Receiver
METHOD PRIVATE CreateMaskReceiver : BOOL
VAR_IN_OUT
	Mask				: RECEIVER_MASK; (* Structure with the information of the bit masks *)
END_VAR
VAR_OUTPUT
	hReceiver			: CAA.HANDLE; (* A valid handle to the Area Receiver *)
	eError				: ERROR; (* Error codes *)
END_VAR
VAR
	eErrorInternal		: CL2.ERROR; (* error codes from the CL2 library *)
END_VAR
IF _hDriver <> CAA.gc_hINVALID THEN
	hReceiver := CL2.CreateMaskReceiver(
					hDriver:= _hDriver, 
					cobIdValue := Mask.dwIdValue, 
					cobIdMask := Mask.dwIdMask, 
					xRTRValue := Mask.xRTRValue, 
					xRTRMask := Mask.xRTRMask, 
					x29BitIdValue := Mask.x29BitIdValue, 
					x29BitIdMask := Mask.x29BitIdMask, 
					xTransmitValue := Mask.xTransmitValue, 
					xTransmitMask := Mask.xTransmitMask, 
					xAlwaysNewest := Mask.xAlwaysNewest, 
					eEvent := CB.EVENT.NO_EVENT, 
					xEnableSyncWindow := FALSE, 
					peError := ADR(eErrorInternal));

	IF (eErrorInternal <> CL2.ERROR.NO_ERROR) THEN
		CL2._DeleteReceiver(hReceiverID:= hReceiver);
		hReceiver:= CAA.gc_hINVALID;
		
		eError:= ERROR.INTERNAL_ERROR;
		
		CreateMaskReceiver:= FALSE;
	ELSE
		CreateMaskReceiver:= TRUE;
	END_IF
ELSE
	eError:= ERROR.NO_CANBUS_DRIVER;
END_IF
END_METHOD

/// Create and Register a IdAreaReceiver. 
METHOD PRIVATE CreateAreaReceiver : BOOL
VAR_INPUT
	hDriver			: CAA.HANDLE; (* Handle to the CANBus Driver *)
END_VAR
VAR_IN_OUT
	ReceiverArea	: RECEIVER_AREA; (* Structure with the information of the bit masks and a range of CAN-ID *)
END_VAR
VAR
	eErrorInternal	: CL2.ERROR; (* error codes from the CL2 library *)
END_VAR
VAR_OUTPUT
	hReceiver		: CAA.HANDLE; (* A valid handle to the Area Receiver *)
	eError			: ERROR; (* Error codes *)
END_VAR
IF hDriver <> CAA.gc_hINVALID THEN
	IF hReceiver = CAA.gc_hINVALID THEN
		hReceiver:= CL2.CreateIdAreaReceiver(
				hDriver:= hDriver, 
				xAlwaysNewest:= FALSE, 
				eEvent:= CB.EVENT.NO_EVENT, 
				xEnableSyncWindow:= FALSE, 
				peError:= ADR(eErrorInternal));
		IF eErrorInternal = CL2.ERROR.NO_ERROR THEN
			IF ReceiverArea.dwIdStart < ReceiverArea.dwIdEnd THEN
				eErrorInternal:= CL2.RegisterIdArea(
						hReceiverID:= hReceiver, 
						cobIdStart:= ReceiverArea.dwIdStart, 
						cobIdEnd:= ReceiverArea.dwIdEnd, 
						xRTRValue:= ReceiverArea.xRTRValue, 
						xRTRMask:= ReceiverArea.xRTRMask, 
						x29BitIdValue:= FALSE, 
						x29BitIdMask:= TRUE, 
						xTransmitValue:= ReceiverArea.xTransmitValue, 
						xTransmitMask:= ReceiverArea.xTransmitMask);
				IF eErrorInternal <> CL2.ERROR.NO_ERROR THEN
					hReceiver:= CAA.gc_hINVALID;
					eError:= ERROR.INTERNAL_ERROR;
				ELSE
					eError:= ERROR.NO_ERROR;
					CreateAreaReceiver:= TRUE;
				END_IF
			ELSE
				eError:= ERROR.START_VALUE_GT_END;
				
			END_IF
		ELSE
			eError:= ERROR.INTERNAL_ERROR;			
		END_IF
	END_IF	
ELSE
	eError:= ERROR.NO_CANBUS_DRIVER;
END_IF
END_METHOD

/// ReceiveMessage expects a valid handle to either an AreaReceiver or a MaskReceiver. With receivers it is
/// possible to filter incoming messages.
/// If a time limit is set, the receiver will only receive messages until the time is up. 
/// It there was no time limit set (tTimeLimit:= 0), the receiver receives messages until the time for the cycle is up.
/// This may cause a lock on the driver.
/// Received messages will be passed to the Message Processor. All message information will be available there.
/// The Message Processor must be implemented by the user.
METHOD PRIVATE ReceiveQueued : BOOL
VAR_INPUT
	hReceiver 		: CAA.HANDLE; (* Eather a MaskReceiver or AreaReceiver *)
	itfMsgProcessor : IMessageProcessor; (* The Message Processor will process the read messages accrding to the implementation of the user *)
	tTimeLimit		: TIME; (* The TimeLimit sets the limit for reading messages in one cycle *)
END_VAR
VAR_OUTPUT
	eError			: ERROR; (* Error codes *)
END_VAR
VAR
	eErrorInternal	: CL2.ERROR; (* error codes from the CL2 library *)
	hMessage		: CAA.HANDLE := CAA.gc_hINVALID; (* Handle for an incoming message *)
	Message			: RxMESSAGE;
	pData			: POINTER TO CL2i.DATA; (* Pointer to the data-array of the incoming message *)
	ctMsgLeft		: CAA.COUNT; (* Counter of the messages left in the queue *)
	i				: INT; (* counter variable *)
	xWatchdog		: BOOL; 
	timeout			: TON;
	udiTSP			: UDINT; (* Only if the driver supports TimeStamps. If not the value is 0. Compare TimeStamp by calling SysTimeGetUs() function *)
END_VAR
IF tTimeLimit > T#0MS THEN 
	xWatchdog := TRUE;
END_IF

REPEAT
	IF xWatchdog THEN
		timeout(IN:= TRUE, PT:= tTimeLimit);
	END_IF
	
	hMessage:= CL2.Read(hReceiverID:= hReceiver, pctMsgLeft:= ADR(ctMsgLeft), peError:= ADR(eErrorInternal));
	/// If a message was received the frame information and the data-array will be written into Message.
	IF hMessage <> CAA.gc_hINVALID THEN			
		Message.udiCanId:= CL2.GetMessageId(hMessage:= hMessage, peError:= ADR(eErrorInternal));
		Message.usiDataLength:= CL2.GetMessageLength(hMessage:= hMessage, peError:= ADR(eErrorInternal));
		Message.xRTR:= CL2.IsRTRMessage(hMessage:= hMessage, peError:= ADR(eErrorInternal));
		Message.xIs29BitMessage:= CL2.Is29BitIdMessage(hMessage:= hMessage, peError:= ADR(eErrorInternal));
		Message.xIsTxMessage:= CL2.IsTransmitMessage(hMessage:= hMessage, peError:= ADR(eErrorInternal));
		udiTSP:= CL2.GetTimeStamp(hMessage:= hMessage, peError:= ADR(eErrorInternal));
		IF Message.usiDataLength > 0 THEN
			pData:= CL2.GetMessageDataPointer(hMessage:= hMessage, peError:= ADR(eErrorInternal));	
		
			IF (pData <> CAA.gc_pNULL) THEN
				FOR i:= 0 TO Message.usiDataLength - 1 DO
					Message.abyData[i] := pData^[i];
				END_FOR
			END_IF
		END_IF
		
		/// The received message will be processed by the Message Processor
		itfMsgProcessor.ProcessMessage(Message:= Message);
		ReceiveQueued := TRUE;
	ELSIF eErrorInternal <> CL2.ERROR.NO_ERROR THEN
		eError:= ERROR.INTERNAL_ERROR;
	END_IF
	
	/// When finished processing the data the memory for the message handle hMessage will be freed by calling CL2.FreeMessage()		
	CL2.FreeMessage(hMessage := hMessage);
UNTIL timeout.Q OR (ctMsgLeft = 0)
END_REPEAT
END_METHOD

/// Create a Single ID Receiver
METHOD PRIVATE CreateSingleIDReceiver : BOOL
VAR_INPUT
	hDriver			: CAA.HANDLE; (* Handle to the CANBus Driver *)
	canId			: UDINT; (* canId to receive *)
	xRTR			: BOOL; (* remote transmission request *)
	x29BitId		: BOOL; (* 29bit CAN-ID *)
	xTransmit		: BOOL; (* bit sign of feedback *)
	xAlwaysNewest	: BOOL; (* TRUE: only the newest message is stored; FALSE: all received messages are stored in chronological order *)
	
END_VAR
VAR_OUTPUT
	hReceiver		: CAA.HANDLE; (* A valid handle to the Area Receiver *)
	eError			: ERROR; (* Error codes *)
END_VAR
VAR
	eErrorInternal	: CL2.ERROR; (* error codes from the CL2 library *)
END_VAR
IF hDriver <> CAA.gc_hINVALID THEN
	hReceiver:= CL2.CreateSingleIdReceiver(
		hDriver:= hDriver, 
		cobId:= canId, 
		xRTR:= xRTR, 
		x29BitId:= x29BitId, 
		xTransmit:= xTransmit, 
		xAlwaysNewest:= xAlwaysNewest, 
		eEvent:= CB.EVENT.NO_EVENT, 
		xEnableSyncWindow:= FALSE, 
		peError:= ADR(eErrorInternal));
		IF eErrorInternal <> CL2.ERROR.NO_ERROR THEN
			eError:= ERROR.INTERNAL_ERROR;
		END_IF
ELSE
	eError:= ERROR.NO_CANBUS_DRIVER;
END_IF
END_METHOD

/// This Private Method creates an CANbus driver by useing the information of DRIVER_CONFIG.
/// After the driver creation was completed a handle to the driver will be returned. 
METHOD PRIVATE CreateDriver : BOOL
VAR_INPUT
	x29bitSupport	: BOOL;
END_VAR
VAR_IN_OUT
	DriverConfig	: DRIVER_CONFIG; (* This structure contains the informaiton for creating a CANbus Driver *)	
END_VAR
VAR_OUTPUT
	hDriver			: CAA.HANDLE; (* A handle to the created CANbus Driver *)
	eError			: ERROR; (* Error codes *)
END_VAR
VAR
	eErrorInternal	: CL2.ERROR; (* error codes from the CL2 library *)
END_VAR
/// If there is not jet a CANbus Driver one will be created with CL2.DriverOpenH()
IF hDriver = CAA.gc_hINVALID THEN
	hDriver:= CL2.DriverOpenH(
			usiNetId:= DriverConfig.usiNetwork, 
			uiBaudrate:= DriverConfig.uiBaudrate, 
			xSupport29Bits:= x29bitSupport, 
			ctMessages:= DriverConfig.ctMessages, 
			peError:= ADR(eErrorInternal));
	
	/// In case an error occured when the driver was created, the driver will be cloese, all pointers set to NULL, 
	/// an error code will be set and the function returnes FALSE 						
	IF (eErrorInternal <> CL2.ERROR.NO_ERROR) THEN
		IF hDriver <> CAA.gc_hINVALID THEN
			CL2.DriverClose(hDriver:= hDriver);
		END_IF
		hDriver:= CAA.gc_hINVALID;
		IF (eErrorInternal = CL2.ERROR.NO_DRIVER) THEN
			eError:= ERROR.CANBUS_DRIVER_NOT_CREATED;
		ELSIF (eErrorInternal = CL2.ERROR.WRONG_BAUDRATE) THEN
			eError:= ERROR.WRONG_BAUDRATE;
		ELSIF (eErrorInternal = CL2.ERROR.NO_29BIT_ID) THEN
			eError:= ERROR.ONLY_11BIT_CANID_ALLOWED;
		ELSIF (eErrorInternal = CL2.ERROR.WRONG_PARAM) THEN
			eError:= ERROR.WRONG_PARAMETER;
		ELSE			
			eError:= ERROR.INTERNAL_ERROR;
		END_IF
	ELSE
	/// In case the driver creation was succesful the Method outputs a valid handle of the driver and 
	/// sets its return value to TRUE
		CreateDriver:= TRUE;
	END_IF
END_IF
END_METHOD

PROPERTY BusAlarm : BOOL
GET
BusAlarm:= CL2.GetBusAlarm(hDriver:= _hDriver, peError:=ADR(_eErrorInternal) );
END_GET
END_PROPERTY

/// Creates a receiver to receive messages within a range of CAN-IDs.
/// It is also possible to use and the same CAN-ID as Start and End value.
METHOD GetAreaReceiver : CAA.HANDLE
VAR_IN_OUT
	Area				: RECEIVER_AREA; (* Structure with the information of the bit masks and a range of CAN-IDs *)
END_VAR
VAR_OUTPUT
	eError				: ERROR; (* Error codes *)
END_VAR
VAR
	hReceiverInfo		: CAA.HANDLE;
	pReceiverInfo		: POINTER TO RECEIVER_INFO;
END_VAR
IF _hDriver <> CAA.gc_hINVALID THEN
	/// In case the CAN-ID Start and the CAN-ID End are identical a receiver for a single CAN-ID will automatically be created.
	IF area.dwIdStart > 2047 OR area.dwIdEnd > 2047 THEN
		eError := ERROR.ONLY_11BIT_CANID_ALLOWED;
	ELSE
		hReceiverInfo := GetReceiverBlock(peError := ADR(eError), pReceiverInfo => pReceiverInfo);
		IF pReceiverInfo <> CAA.gc_pNULL THEN
			IF Area.dwIdStart = Area.dwIdEnd THEN
				 CreateSingleIDReceiver(hDriver:= _hDriver, canId:= Area.dwIdStart, xRTR:= Area.xRTRValue, 
										x29BitId:= FALSE, xTransmit:= Area.xTransmitValue, xAlwaysNewest:= FALSE, 
										hReceiver=> pReceiverInfo^.hReceiver, eError=> eError);
			ELSE
				/// Creates a receiver for messages within a range of CAN-IDs.
				CreateAreaReceiver(hDriver:= _hDriver, ReceiverArea:= Area, hReceiver=> pReceiverInfo^.hReceiver, eError=> eError);
			END_IF
			
			IF pReceiverInfo^.hReceiver <> CAA.gc_hINVALID THEN
				pReceiverInfo^.eType := RECEIVERTYPE.QUEUED_RECEIVER;
				GetAreaReceiver:= hReceiverInfo;
			ELSE
				FreeReceiverBlock(hReceiverInfo);	
			END_IF
		END_IF
	END_IF
ELSE
	eError:= ERROR.NO_CANBUS_DRIVER;
END_IF
END_METHOD

/// Creates a receiver to receive messages according to a specific Bit Mask.
METHOD GetMaskReceiver : CAA.HANDLE
VAR_IN_OUT
	Mask				: RECEIVER_MASK; (* Structure with the information of the bit masks *)
END_VAR
VAR_OUTPUT
	eError				: ERROR; (* Error codes *)
END_VAR
VAR
	hReceiverInfo		: CAA.HANDLE;
	pReceiverInfo		: POINTER TO RECEIVER_INFO;
END_VAR
IF _hDriver <> CAA.gc_hINVALID THEN
	hReceiverInfo := GetReceiverBlock(peError := ADR(eError), pReceiverInfo => pReceiverInfo);
	IF pReceiverInfo <> CAA.gc_pNULL THEN
		CreateMaskReceiver(Mask:= Mask, hReceiver=> pReceiverInfo^.hReceiver, eError=> eError);
		IF pReceiverInfo^.hReceiver <> CAA.gc_hINVALID THEN
			IF Mask.xAlwaysNewest THEN
				pReceiverInfo^.eType := RECEIVERTYPE.ALWAYS_NEWEST_RECEIVER;
			ELSE
				pReceiverInfo^.eType := RECEIVERTYPE.QUEUED_RECEIVER;
			END_IF
			GetMaskReceiver:= hReceiverInfo;
		ELSE
			FreeReceiverBlock(hReceiverInfo);	
		END_IF
	END_IF
ELSE
	eError:= ERROR.NO_CANBUS_DRIVER;
END_IF
END_METHOD

/// ReceiveMessage expects a valid handle to either an AreaReceiver or a MaskReceiver. With receivers it is
/// possible to filter incoming messages.
/// If a time limit is set, the receiver will only receive messages until the time is up. 
/// It there was no time limit set (tTimeLimit:= 0), the receiver receives messages until the time for the cycle is up.
/// This may cause a lock on the driver.
/// Received messages will be passed to the Message Processor. All message information will be available there.
/// The Message Processor must be implemented by the user.
METHOD ReceiveMessage : BOOL
VAR_INPUT
	hReceiver 		: CAA.HANDLE; (* Either a MaskReceiver or AreaReceiver *)
	itfMsgProcessor : IMessageProcessor; (* The Message Processor will process the read messages accrding to the implementation of the user *)
	tTimeLimit		: TIME; (* The TimeLimit sets the limit for reading messages in one cycle *)
END_VAR
VAR_OUTPUT
	eError			: ERROR; (* Error codes *)
END_VAR
VAR
	eErrorInternal	: CL2.ERROR; (* error codes from the CL2 library *)
	hMessage		: CAA.HANDLE := CAA.gc_hINVALID; (* Handle for an incoming message *)
	Message			: RxMESSAGE;
	pData			: POINTER TO CL2i.DATA; (* Pointer to the data-array of the incoming message *)
	ctMsgLeft		: CAA.COUNT; (* Counter of the messages left in the queue *)
	i				: INT; (* counter variable *)
	xWatchdog		: BOOL; 
	timeout			: TON;
	udiTSP			: UDINT; (* Only if the driver supports TimeStamps. If not the value is 0. Compare TimeStamp by calling SysTimeGetUs() function *)
	pReceiverInfo   : POINTER TO RECEIVER_INFO;
	eMBMError : MBM.ERROR;
END_VAR
IF hReceiver <> CAA.gc_hINVALID THEN
	/// If the time limit is set to T#0 new messages will be received until there are no more messages
	/// in the queue. If a time limit is set, messages will be received until the limit is up.	
	pReceiverInfo := MBM.BlockGetData(hBlock := hReceiver, peError := ADR(eMBMError));
	IF pReceiverInfo <> CAA.gc_pNULL THEN
		IF pReceiverInfo^.eType = RECEIVERTYPE.QUEUED_RECEIVER THEN
			ReceiveMessage := ReceiveQueued(hReceiver := pReceiverInfo^.hReceiver, itfMsgProcessor := itfMsgProcessor, tTimeLimit := tTimeLimit, eError => eError);
		ELSE
			ReceiveMessage := ReceiveAlwaysNewest(hReceiver := pReceiverInfo^.hReceiver, itfMsgProcessor := itfMsgProcessor, eError => eError);
		END_IF
	ELSE
		eError:= ERROR.NO_VALID_RECEIVER;
	END_IF
ELSE
	eError:= ERROR.NO_VALID_RECEIVER;
END_IF
END_METHOD

METHOD FB_Init : BOOL
VAR_INPUT
  bInitRetains : BOOL; // if TRUE, the retain variables are initialized (warm start / cold start)
  bInCopyCode : BOOL;  // if TRUE, the instance afterwards gets moved into the copy code (online change)
END_VAR
VAR
	eMBMError : MBM.ERROR;
END_VAR
_hReceiverPool := MBM.PoolCreateH(ctNumBlocks := 10, szBlockSize := SIZEOF(RECEIVER_INFO), eEmpty := 0, peError := ADR(eMBMError));
END_METHOD

/// This method aggregates diagnostic information in DIAGNOSIS_INFO 
METHOD GetBusDiagnosis : BOOL
VAR_IN_OUT
	DiagnosticInfo		: DIAGNOSIS_INFO; (* This data type descripes diagnostic information  *)
END_VAR
VAR_OUTPUT
	eError				: ERROR; (* Error codes *)
END_VAR
VAR
	eErrorInternal		: CL2.ERROR; (* error codes from the CL2 library *)
END_VAR
IF _hDriver <> CAA.gc_hINVALID THEN
	DiagnosticInfo.ctReceiveCounter:= CL2.GetReceiveCounter(hDriver:= _hDriver,  peError:= ADR(eErrorInternal));
	DiagnosticInfo.ctRxErrorCounter:= CL2.GetReceiveErrorCounter(hDriver:= _hDriver,  peError:= ADR(eErrorInternal));
	DiagnosticInfo.ctSendCounter:= CL2.GetTransmitCounter(hDriver:= _hDriver,  peError:= ADR(eErrorInternal));
	DiagnosticInfo.ctTxErrorCounter:= CL2.GetTransmitErrorCounter(hDriver:= _hDriver,  peError:= ADR(eErrorInternal));
	DiagnosticInfo.eState:= ANY_NUM_TO_BYTE(CL2.GetBusState(hDriver:= _hDriver,  peError:= ADR(eErrorInternal)));
	DiagnosticInfo.uiBaudrate:= CL2.GetBaudrate(hDriver:= _hDriver,  peError:= ADR(eErrorInternal));
	DiagnosticInfo.usiBusLoad:= CL2.GetBusload(hDriver:= _hDriver,  peError:= ADR(eErrorInternal));
	DiagnosticInfo.xSendingActive:= CL2.IsSendingActive(hDriver:= _hDriver,  peError:= ADR(eErrorInternal));
	DiagnosticInfo.xBusAlarm:= CL2.GetBusAlarm(hDriver:= _hDriver,  peError:= ADR(eErrorInternal));
	DiagnosticInfo.ctLostCounter:= CL2.GetLostCounter(hDriver:= _hDriver,  peError:= ADR(eErrorInternal));
	DiagnosticInfo.ctReceivePoolSize:= CL2.GetReceivePoolSize(hDriver:= _hDriver,  peError:= ADR(eErrorInternal));
	DiagnosticInfo.ctReceiveQueueLength:= CL2.GetReceiveQueueLength(hDriver:= _hDriver,  peError:= ADR(eErrorInternal));
	DiagnosticInfo.ctTransmitPoolSize:= CL2.GetTransmitPoolSize(hDriver:= _hDriver,  peError:= ADR(eErrorInternal));
	DiagnosticInfo.ctTransmitQueueLength:= CL2.GetTransmitQueueLength(hDriver:= _hDriver,  peError:= ADR(eErrorInternal));
	
	IF eErrorInternal <> CL2.ERROR.NO_ERROR THEN
		eError:= error.INTERNAL_ERROR;
	ELSE
		GetBusDiagnosis:= TRUE;	
	END_IF

ELSE
	eError:= ERROR.NO_CANBUS_DRIVER;
END_IF
END_METHOD

/// This method resets the CANBus if the driver is in 'bus alarm' state. 
METHOD ResetBusAlarm : BOOL
VAR_INPUT
END_VAR
VAR_OUTPUT
	eError			: ERROR; (* Error codes *)
END_VAR
VAR
	eErrorInternal	: CL2.ERROR; (* error codes from the CL2 library *)
END_VAR
IF _hDriver <> CAA.gc_hINVALID THEN
	eErrorInternal:= CL2.ResetBusAlarm(hDriver:= _hDriver);
	
	IF eErrorInternal <> CL2.ERROR.NO_ERROR THEN
		eError:= ERROR.INTERNAL_ERROR;
	ELSE
		ResetBusAlarm:= TRUE;
	END_IF
ELSE
	eError:= ERROR.NO_CANBUS_DRIVER;
END_IF
END_METHOD

{attribute 'hide'}
PROPERTY Is29bit : BOOL
GET
END_GET
END_PROPERTY

METHOD GetSingleIdReceiver : CAA.HANDLE
VAR_IN_OUT
	(* Structure with the information of the bit masks *)
	SingleId	: RECEIVER_SINGLE_ID;
END_VAR
VAR_OUTPUT
	(* Error codes *)
	eError	: ERROR;
END_VAR
VAR
	hReceiverInfo		: CAA.HANDLE;
	pReceiverInfo		: POINTER TO RECEIVER_INFO;
END_VAR
IF _hDriver <> CAA.gc_hINVALID THEN
	hReceiverInfo := GetReceiverBlock(peError := ADR(eError), pReceiverInfo => pReceiverInfo);
	IF pReceiverInfo <> CAA.gc_pNULL THEN
		CreateSingleIDReceiver(hDriver:= _hDriver, canId:= SingleId.dwCanId, xRTR:= SingleId.xRTRValue, 
								x29BitId:= SingleId.x29BitIdValue, xTransmit:= SingleId.xTransmitValue, xAlwaysNewest:= SingleId.xAlwaysNewest, 
								hReceiver=> pReceiverInfo^.hReceiver, eError=> eError);
		IF pReceiverInfo^.hReceiver <> CAA.gc_hINVALID THEN
			IF SingleId.xAlwaysNewest THEN
				pReceiverInfo^.eType := RECEIVERTYPE.ALWAYS_NEWEST_RECEIVER;
			ELSE
				pReceiverInfo^.eType := RECEIVERTYPE.QUEUED_RECEIVER;
			END_IF
			GetSingleIdReceiver:= hReceiverInfo;
		ELSE
			FreeReceiverBlock(hReceiverInfo);	
		END_IF
	END_IF
ELSE
	eError:= ERROR.NO_CANBUS_DRIVER;
END_IF
END_METHOD

END_FUNCTION_BLOCK

// Function Blocks/Object Oriented Programming/CANBus_29bit
/// | CANBus Function Block 29 Bit can handle frames with 11bit CAN-IDs and 29bit CAN-IDs. 
/// | An instance of this function block has to be created in order for being able to send or receive messages. 
/// | The FB expects a complete structure of the type DRIVER_CONFIG to set up the CANBus. There are two methods 
/// | for sending. SendMessage() will send messages with a standard 11 bit CAN-ID, SendMessage29bit() will send messages 
/// | with a 29 bit CAN-ID. 
FUNCTION_BLOCK CANBus_29bit EXTENDS CANBus_Base IMPLEMENTS ICANBus11bit, ICANBus29bit
VAR_INPUT
END_VAR
VAR_OUTPUT
END_VAR
VAR
END_VAR

/// Call of the CANBus_Base FB
SUPER^._x29bitSupport:=TRUE;
SUPER^();

/// This method resets the CANBus if the driver is in 'bus alarm' state. 
METHOD ResetBusAlarm : BOOL
VAR_INPUT
END_VAR
VAR_OUTPUT
	eError			: ERROR; (* Error codes *)
END_VAR
/// Method call of the CANBus_Base FB
ResetBusAlarm:= SUPER^.ResetBusAlarm(eError=> eError);
END_METHOD

/// Send a message. If the message got sent the return value is true.
METHOD SendMessage : BOOL
VAR_IN_OUT
	Message 		: MESSAGE; (* Message information and data. *)
END_VAR
VAR_OUTPUT
	eError			: ERROR; (* Error codes *)
END_VAR
SendMessage := SUPER^.SendMessage(Message := Message, eError => eError);
END_METHOD

/// Deletes given receiver
METHOD DeleteReceiver : BOOL
VAR_IN_OUT
	hReceiver		: CAA.HANDLE; (* Receiver to be deleted *)
END_VAR
VAR_OUTPUT
	eError			: ERROR; (* Error codes *)
END_VAR
/// Method call of the CANBus_Base FB
DeleteReceiver:= super^.DeleteReceiver(hReceiver:= hReceiver, eError=> eError);
END_METHOD

/// | Creates a mask for receiving messages. (With each call of this function a Receiver is created. 
/// | Therefor the method should not be called cyclic.)
METHOD GetMaskReceiver : CAA.HANDLE
VAR_IN_OUT
	Mask				: RECEIVER_MASK; (* Structure with the information of the bit masks *)
END_VAR
VAR_OUTPUT
	eError				: ERROR; (* Error codes *)
END_VAR
/// Method call of the CANBus_Base FB
GetMaskReceiver:= SUPER^.GetMaskReceiver(Mask:= Mask, eError=> eError);
END_METHOD

/// | ReceiveMessage expects a valid handle to either an AreaReceiver, SingleIdReceiver or a MaskReceiver. 
/// | With receivers it is possible to filter incoming messages. If a time limit is set, the receiver will 
/// | receive in each cycle messages until the time is up. It there is no time limit set (tTimeLimit:= 0), 
/// | the receiver receives messages until the receiver buffer is empty. If the time limit is too small it 
/// | may be that not all received messages are processed and therefor the buffer gets smaller until there 
/// | are no free message handles left. Received messages will be passed to the Message Processor. All message 
/// | information will be available there. The Message Processor must be implemented by the user.
METHOD ReceiveMessage : BOOL
VAR_INPUT
	hReceiver 		: CAA.HANDLE; (* Either a MaskReceiver, SingleIdReceiver or AreaReceiver *)
	itfMsgProcessor : IMessageProcessor; (* The Message Processor will process the read messages accrding to the implementation of the user *)
	tTimeLimit		: TIME; (* The time limit for reading messages. (T#0s means no time limit) *)
END_VAR
VAR_OUTPUT
	eError			: ERROR; (* Error codes *)
END_VAR
/// Method call of the CANBus_Base FB
ReceiveMessage:= SUPER^.ReceiveMessage(hReceiver:= hReceiver, itfMsgProcessor:= itfMsgProcessor, tTimeLimit:= tTimeLimit, eError=> eError);
END_METHOD

{attribute 'hide'}
PROPERTY Is29bit : BOOL
GET
Is29bit:= TRUE;
END_GET
END_PROPERTY

/// Closes the CAN Driver. After closing, messages can't be received or transmitted anymore.
METHOD CloseCANDriver : BOOL
VAR_INPUT
END_VAR
VAR_OUTPUT
	eError			: ERROR; (* Error codes *)
END_VAR
CloseCANDriver:= SUPER^.CloseCANDriver(eError=> eError);
END_METHOD

/// | Creates a receiver to receive messages within a range of CAN-IDs. 
/// | (With each call of this function a Receiver is created. Therefor the method should not be called cyclic.)
METHOD GetAreaReceiver : CAA.HANDLE
VAR_IN_OUT
	Area				: RECEIVER_AREA; (* Structure with the information of the bit masks and a range of CAN-IDs *)
END_VAR
VAR_OUTPUT
	eError				: ERROR; (* Error codes *)
END_VAR
/// Method call of the CANBus_Base FB
GetAreaReceiver:= SUPER^.GetAreaReceiver(Area:= Area, eError=> eError);
END_METHOD

/// This method aggregates diagnostic information in DIAGNOSIS_INFO
METHOD GetBusDiagnosis : BOOL
VAR_IN_OUT
	DiagnosticInfo		: DIAGNOSIS_INFO; (* This data type describes diagnostic information *)
END_VAR
VAR_OUTPUT
	eError				: ERROR; (* Error codes *)
END_VAR
/// Method call of the CANBus_Base FB
GetBusDiagnosis:= SUPER^.GetBusDiagnosis(DiagnosticInfo:= DiagnosticInfo, eError=> eError);
END_METHOD

/// | Generates a receiver for filtering a single CanId. (With each call of this function a 
/// | Receiver is created. Therefor the method should not be called cyclic.)
METHOD GetSingleIdReceiver : CAA.HANDLE
VAR_IN_OUT
	(* Structure with the information of the bit masks *)
	SingleId	: RECEIVER_SINGLE_ID;
END_VAR
VAR_OUTPUT
	(* Error codes *)
	eError	: ERROR;
END_VAR
/// Method call of the CANBus_Base FB
GetSingleIdReceiver:= SUPER^.GetSingleIdReceiver(SingleId:= SingleId, eError=> eError);
END_METHOD

END_FUNCTION_BLOCK

// Interfaces/ICANBus11bit
{attribute 'hide'}
INTERFACE ICANBus11bit EXTENDS ICANBusBase

END_INTERFACE

// Function Blocks/Graphical Programming/CANDriver_29bit
/// | This CAN Driver can handle frames with 29bit CAN-IDs and 11bit CAN-IDs. If a CAN Sender gets instantiated with this Driver, messages
/// | will be sent ether as 11 bit or 29 bit frames, depending on the xSendAs29bitMsg flag of MESSAGE. If the flag is TRUE, messages
/// | are sent as 29bit frame. Any Receiver instantiated with this Driver can receive 11 bit and 29 bit CAN-ID frames.  
FUNCTION_BLOCK CANDriver_29bit EXTENDS CBM.LTrig IMPLEMENTS ICANDriver
VAR_INPUT
	xResetBusAlarm	: BOOL; (* TRUE: Reset the Bus Alarm (applies only if the Bus Driver is in alarm state). *)
END_VAR
VAR_IN_OUT
	DriverConfig	: DRIVER_CONFIG; (* Information to setup the CANbus Driver *)
END_VAR
VAR_OUTPUT
	xBusAlarm		: BOOL; (* indicates if a Bus Alarm occurred *)
	eError			: ERROR; (* Error codes *)
END_VAR
VAR
	_CANBus			: CANBus_29bit;
	_pDriverConfig	: POINTER TO DRIVER_CONFIG;
END_VAR

_pDriverConfig := ADR(DriverConfig);
SUPER^();
IF iError = CBM.ERROR.TIME_OUT THEN
	eError := ERROR.TIME_OUT;
END_IF

{attribute 'hide'}
PROPERTY ICANBus : ICANBusBase
GET
ICANBus:= _CANBus;
END_GET
END_PROPERTY

{attribute 'hide'}
METHOD prvCyclicAction : BOOL
VAR_INPUT
END_VAR
VAR
END_VAR
IF xEnable AND _pDriverConfig <> CAA.gc_pNULL THEN
	_CANBus(DriverConfig:= _pDriverConfig^, eError=> eError);
	IF _CANBus.BusAlarm THEN 
		eError:= ERROR.BUS_ALARM;
		xBusAlarm:= TRUE;
	ELSIF _CANBus.BusAlarm AND xResetBusAlarm  THEN
		_CANBus.ResetBusAlarm(eError=> eError);
		xBusAlarm:= FALSE;
	END_IF
END_IF

IF eError <> ERROR.NO_ERROR THEN
	iError:= 2;
END_IF
END_METHOD

{attribute 'hide'}
METHOD prvResetOutputs : BOOL
VAR_INPUT
END_VAR
VAR
END_VAR
eError:= ERROR.NO_ERROR;
xBusAlarm:= FALSE;
SUPER^.prvResetOutputs();
END_METHOD

{attribute 'hide'}
METHOD prvStart : BOOL
VAR_INPUT
END_VAR
VAR
END_VAR
END_METHOD

{attribute 'hide'}
METHOD prvAbort : BOOL
VAR_INPUT
END_VAR
VAR
END_VAR
IF xError THEN (* abort because of error *)
	_CANBus.CloseCANDriver(eError=> eError);
ELSE
	_CANBus.CloseCANDriver(eError=> eError);
END_IF
xAbortInProgress:= FALSE;
END_METHOD

END_FUNCTION_BLOCK

// Function Blocks/Graphical Programming/CANMaskReceiver
/// | This receives messages according to a specific Bit Mask. If a time limit is set, the receiver will receive 
/// | in each cycle messages until the time is up. It there is no time limit set (tTimeLimit:= 0), 
/// | the receiver receives messages until the receiver buffer is empty. If the time limit is too small it 
/// | may be that not all received messages are processed and therefor the buffer gets smaller until there are no 
/// | free message handles left. Received messages will be passed to the Message Processor. 
/// | All message information will be available there. The Message Processor must be implemented by the user.
FUNCTION_BLOCK CANMaskReceiver EXTENDS CBM.LTrig
VAR_INPUT
	itfCANDriver		: ICANDriver; (* An Mask Receiver will be created for this CAN Driver *)
	itfMsgProcessor		: IMessageProcessor; (* Processed the message information. The user must implement the Message Processor. *)
	tTimeLimit			: TIME; (* The time limit for reading messages. (T#0s means no time limit) *)
END_VAR
VAR_IN_OUT
	Mask				: RECEIVER_MASK; (* Filter criteria for the receiver *)
END_VAR
VAR_OUTPUT
	eError				: ERROR; (* Error codes *)
END_VAR
VAR
	_hReceiver			: CAA.HANDLE; (* The receiver *)
	_pMask				: POINTER TO RECEIVER_MASK;
END_VAR

_pMask := ADR(Mask);
SUPER^();
IF iError = CBM.ERROR.TIME_OUT THEN
	eError := ERROR.TIME_OUT;
END_IF

{attribute 'hide'}
METHOD prvStart : BOOL
VAR_INPUT
END_VAR
VAR
END_VAR
END_METHOD

{attribute 'hide'}
METHOD prvAbort : BOOL
VAR_INPUT
END_VAR
VAR
END_VAR
IF _hReceiver <> CAA.gc_hINVALID THEN
	itfCANDriver.ICANBus.DeleteReceiver(hReceiver:= _hReceiver, eError=> eError);
	_hReceiver := CAA.gc_hINVALID;
END_IF

xAbortInProgress:= FALSE;
END_METHOD

{attribute 'hide'}
METHOD prvCyclicAction : BOOL
VAR_INPUT
END_VAR
VAR
END_VAR
IF xEnable THEN
	IF _hReceiver = CAA.gc_hINVALID AND _pMask <> CAA.gc_pNULL THEN
		_hReceiver:= itfCANDriver.ICANBus.GetMaskReceiver(Mask:= _pMask^, eError=> eError);
	END_IF
	IF eError = ERROR.NO_ERROR THEN	
		itfCANDriver.ICANBus.ReceiveMessage(hReceiver:= _hReceiver, itfMsgProcessor:= itfMsgProcessor, tTimeLimit:= tTimeLimit, eError=> eError);
	END_IF
END_IF

IF eError <> ERROR.NO_ERROR THEN
	iError:= 2;
END_IF
END_METHOD

{attribute 'hide'}
METHOD prvResetOutputs : BOOL
VAR_INPUT
END_VAR
VAR
END_VAR
eError:= ERROR.NO_ERROR;
SUPER^.prvResetOutputs();
END_METHOD

END_FUNCTION_BLOCK

// Function Blocks/Graphical Programming/CANAreaReceiver
/// | This receives messages for a range of CAN-IDs. Please note that the Area Receiver only allows 11bit CAN-IDs. 
/// | If a time limit is set, the receiver will receive in each cycle messages until the time is up. 
/// | It there is no time limit set (tTimeLimit:= 0), the receiver receives messages until the receiver buffer is empty. 
/// | If the time limit is too small it may be that not all received messages are processed and therefore 
/// | the buffer gets smaller until there are no free message handles left. Received messages will be passed to 
/// | the Message Processor. All message information will be available there. 
/// | The Message Processor must be implemented by the user.
FUNCTION_BLOCK CANAreaReceiver EXTENDS CBM.LTrig
VAR_INPUT
	itfCANDriver		: ICANDriver; (* An Area Receiver will be created for this CAN Driver *)
	itfMsgProcessor		: IMessageProcessor; (* Processed the message information. The user must implement the Message Processor. *)
	tTimeLimit			: TIME; (* The time limit for reading messages. (T#0s means no time limit) *)
END_VAR
VAR_IN_OUT
	Area				: RECEIVER_AREA; (* Filter criteria for the receiver *)
END_VAR
VAR_OUTPUT
	eError				: ERROR; (* Error codes *)
END_VAR
VAR
	_hReceiver			: CAA.HANDLE; (* The receiver *)
	_pArea				: POINTER TO RECEIVER_AREA;
END_VAR

_pArea := ADR(Area);
SUPER^();
IF iError = CBM.ERROR.TIME_OUT THEN
	eError := ERROR.TIME_OUT;
END_IF

{attribute 'hide'}
METHOD prvAbort : BOOL
VAR_INPUT
END_VAR
VAR
END_VAR
IF _hReceiver <> CAA.gc_hINVALID THEN
	itfCANDriver.ICANBus.DeleteReceiver(hReceiver:= _hReceiver, eError=> eError);
	_hReceiver := CAA.gc_hINVALID;
END_IF
xAbortInProgress:= FALSE;
END_METHOD

{attribute 'hide'}
METHOD prvCyclicAction : BOOL
VAR_INPUT
END_VAR
VAR
END_VAR
IF xEnable THEN
	IF _hReceiver = CAA.gc_hINVALID AND _pArea <> CAA.gc_pNULL THEN
		_hReceiver:= itfCANDriver.ICANBus.GetAreaReceiver(Area:= _pArea^, eError=> eError);
	END_IF
	IF eError = ERROR.NO_ERROR THEN
		itfCANDriver.ICANBus.ReceiveMessage(hReceiver:= _hReceiver, itfMsgProcessor:= itfMsgProcessor, tTimeLimit:= tTimeLimit, eError=> eError);
	END_IF
END_IF

IF eError <> ERROR.NO_ERROR THEN
	iError:= 2;
END_IF
END_METHOD

{attribute 'hide'}
METHOD prvResetOutputs : BOOL
VAR_INPUT
END_VAR
VAR
END_VAR
eError:= ERROR.NO_ERROR;
SUPER^.prvResetOutputs();
END_METHOD

{attribute 'hide'}
METHOD prvStart : BOOL
VAR_INPUT
END_VAR
VAR
END_VAR
END_METHOD

END_FUNCTION_BLOCK

// Function Blocks/Graphical Programming/CANBusDiagnosis
/// | CAN Bus Diagnosis delivers a structure of diagnostic information about a CAN Bus Driver.
FUNCTION_BLOCK CANBusDiagnosis EXTENDS CBM.LTrig
VAR_INPUT
	itfCANDriver		: ICANDriver; (* Information will be retrieved from this CAN Driver *)
END_VAR
VAR_IN_OUT
	DiagnosticInfo		: DIAGNOSIS_INFO; (* Describes the diagnostic information  *)
END_VAR
VAR_OUTPUT
	eError				: ERROR; (* Error codes *)
END_VAR
VAR
	_pDiagnosticInfo		: POINTER TO DIAGNOSIS_INFO;
END_VAR

_pDiagnosticInfo := ADR(DiagnosticInfo);
SUPER^();
IF iError = CBM.ERROR.TIME_OUT THEN
	eError := ERROR.TIME_OUT;
END_IF

{attribute 'hide'}
METHOD prvResetOutputs : BOOL
VAR_INPUT
END_VAR
VAR
END_VAR
eError:= ERROR.NO_ERROR;
SUPER^.prvResetOutputs();
END_METHOD

{attribute 'hide'}
METHOD prvCyclicAction : BOOL
VAR_INPUT
END_VAR
VAR
END_VAR
IF xEnable AND _pDiagnosticInfo <> CAA.gc_pNULL THEN
	itfCANDriver.ICANBus.GetBusDiagnosis(DiagnosticInfo:= _pDiagnosticInfo^, eError=> eError);
END_IF

IF eError <> ERROR.NO_ERROR THEN
	iError:= 2;
END_IF
END_METHOD

{attribute 'hide'}
METHOD prvStart : BOOL
VAR_INPUT
END_VAR
VAR
END_VAR
END_METHOD

{attribute 'hide'}
METHOD prvAbort : BOOL
VAR_INPUT
END_VAR
VAR
END_VAR
xAbortInProgress:= FALSE;
END_METHOD

END_FUNCTION_BLOCK

// Function Blocks/Graphical Programming/CANSingleIdReceiver
/// | Generates a receiver for filtering a single CanId. If a time limit is set, the receiver will receive in each cycle 
/// | messages until the time is up. It there is no time limit set (tTimeLimit:= 0), the receiver receives messages 
/// | until the receiver buffer is empty. If the time limit is too small it may be that not all received messages 
/// | are processed and therefor the buffer gets smaller until there are no free message handles left. 
/// | Received messages will be passed to the Message Processor. All message information will be available there. 
/// | The Message Processor must be implemented by the user.
FUNCTION_BLOCK CANSingleIdReceiver EXTENDS CBM.LTrig
VAR_INPUT
	itfCANDriver		: ICANDriver; (* An Area Receiver will be created for this CAN Driver *)
	itfMsgProcessor		: IMessageProcessor; (* Processed the message information. The user must implement the Message Processor. *)
	tTimeLimit			: TIME; (* The time limit for reading messages. (T#0s means no time limit) *)
END_VAR
VAR_IN_OUT
	SingleId			: RECEIVER_SINGLE_ID; (* Filter criteria for the receiver *)
END_VAR
VAR_OUTPUT
	eError				: ERROR; (* Error codes *)
END_VAR
VAR
	_hReceiver			: CAA.HANDLE; (* The receiver *)
	_pSingleId			: POINTER TO RECEIVER_SINGLE_ID;
END_VAR

_pSingleId := ADR(SingleId);
SUPER^();
IF iError = CBM.ERROR.TIME_OUT THEN
	eError := ERROR.TIME_OUT;
END_IF

{attribute 'hide'}
METHOD prvResetOutputs : BOOL
VAR_INPUT
END_VAR
VAR
END_VAR
eError:= ERROR.NO_ERROR;
SUPER^.prvResetOutputs();
END_METHOD

{attribute 'hide'}
METHOD prvStart : BOOL
VAR_INPUT
END_VAR
VAR
END_VAR
END_METHOD

{attribute 'hide'}
METHOD prvAbort : BOOL
VAR_INPUT
END_VAR
VAR
END_VAR
IF _hReceiver <> CAA.gc_hINVALID THEN
	itfCANDriver.ICANBus.DeleteReceiver(hReceiver:= _hReceiver, eError=> eError);
	_hReceiver := CAA.gc_hINVALID;
END_IF
xAbortInProgress:= FALSE;
END_METHOD

{attribute 'hide'}
METHOD prvCyclicAction : BOOL
VAR_INPUT
END_VAR
VAR
END_VAR
IF xEnable THEN
	IF _hReceiver = CAA.gc_hINVALID AND _pSingleId <> CAA.gc_pNULL THEN
		_hReceiver:= itfCANDriver.ICANBus.GetSingleIdReceiver(SingleId:= _pSingleId^ , eError=> eError);
	END_IF
	IF eError = ERROR.NO_ERROR THEN
		itfCANDriver.ICANBus.ReceiveMessage(hReceiver:= _hReceiver, itfMsgProcessor:= itfMsgProcessor, tTimeLimit:= tTimeLimit, eError=> eError);
	END_IF
END_IF

IF eError <> ERROR.NO_ERROR THEN
	iError:= 2;
END_IF
END_METHOD

END_FUNCTION_BLOCK
